% RSLogix 500 project I2P Job 13 B Alexander_Loynd.RSS, saved by version 10.00.00.00 %
PROJECT "ML06A"    % processor: Bul.1763 MicroLogix 1100 Series B %

PROGRAM FILES
  LAD 2   13 rungs

DATA FILES
  O0 OUTPUT  4 elements
  I1 INPUT  6 elements
  S2 STATUS  66 elements
  B3 BINARY  1 elements
  T4 TIMER  1 elements
  C5 COUNTER  1 elements
  R6 CONTROL  1 elements
  N7 INTEGER  1 elements
  F8 FLOAT  1 elements

LADDER 2
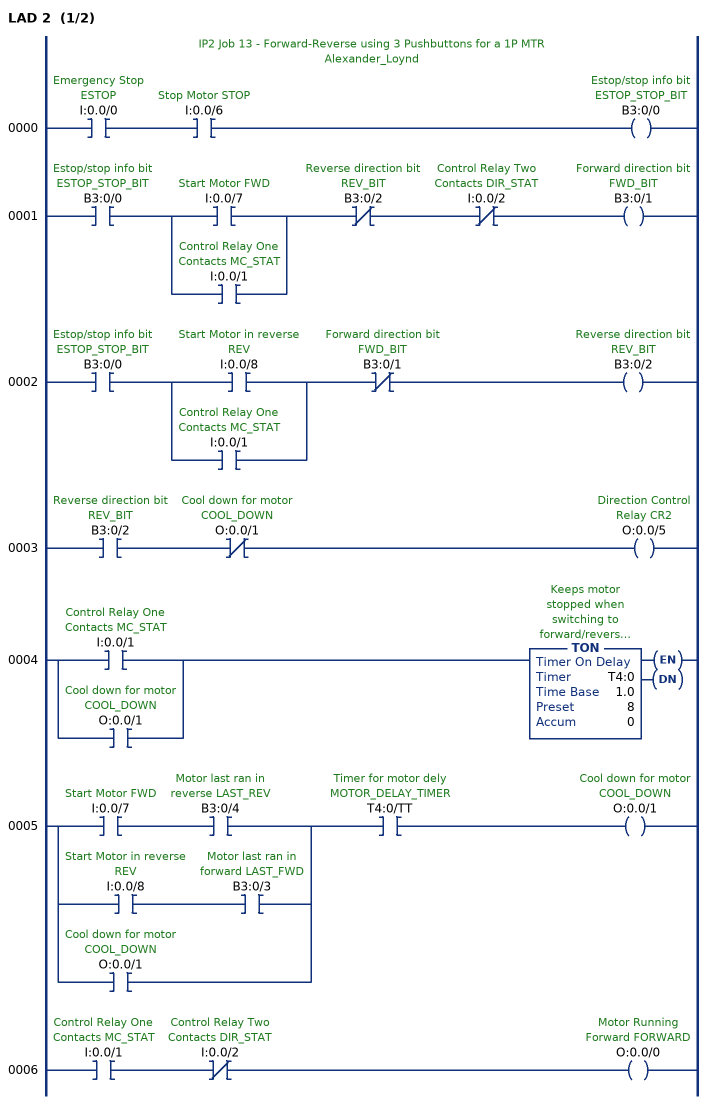
% Rung: 0 %
% IP2 Job 13 - Forward-Reverse using 3 Pushbuttons for a 1P MTR
% Alexander_Loynd %
SOR XIC I:0.0/0 XIC I:0.0/6 OTE B3:0/0 EOR
%   I:0.0/0  ESTOP  "Emergency Stop" %
%   I:0.0/6  STOP  "Stop Motor" %
%   B3:0/0  ESTOP_STOP_BIT  "Estop/stop info bit" %
% Rung: 1 %
SOR XIC B3:0/0 BST XIC I:0.0/7 NXB XIC I:0.0/1 BND XIO B3:0/2 XIO I:0.0/2 OTE B3:0/1 EOR
%   B3:0/0  ESTOP_STOP_BIT  "Estop/stop info bit" %
%   I:0.0/7  FWD  "Start Motor" %
%   I:0.0/1  MC_STAT  "Control Relay One Contacts" %
%   B3:0/2  REV_BIT  "Reverse direction bit" %
%   I:0.0/2  DIR_STAT  "Control Relay Two Contacts" %
%   B3:0/1  FWD_BIT  "Forward direction bit" %
% Rung: 2 %
SOR XIC B3:0/0 BST XIC I:0.0/8 NXB XIC I:0.0/1 BND XIO B3:0/1 OTE B3:0/2 EOR
%   B3:0/0  ESTOP_STOP_BIT  "Estop/stop info bit" %
%   I:0.0/8  REV  "Start Motor in reverse" %
%   I:0.0/1  MC_STAT  "Control Relay One Contacts" %
%   B3:0/1  FWD_BIT  "Forward direction bit" %
%   B3:0/2  REV_BIT  "Reverse direction bit" %
% Rung: 3 %
SOR XIC B3:0/2 XIO O:0.0/1 OTE O:0.0/5 EOR
%   B3:0/2  REV_BIT  "Reverse direction bit" %
%   O:0.0/1  COOL_DOWN  "Cool down for motor" %
%   O:0.0/5  CR2  "Direction Control Relay" %
% Rung: 4 %
SOR BST XIC I:0.0/1 NXB XIC O:0.0/1 BND TON T4:0 1.0 8 0 EOR
%   I:0.0/1  MC_STAT  "Control Relay One Contacts" %
%   O:0.0/1  COOL_DOWN  "Cool down for motor" %
%   T4:0  MTR_DELAY  "Keeps motor stopped when switching to forward/reverse" %
% Rung: 5 %
SOR BST XIC I:0.0/7 XIC B3:0/4 NXB BST XIC I:0.0/8 XIC B3:0/3 NXB XIC O:0.0/1 BND BND XIC T4:0/TT OTE O:0.0/1 EOR
%   I:0.0/7  FWD  "Start Motor" %
%   B3:0/4  LAST_REV  "Motor last ran in reverse" %
%   I:0.0/8  REV  "Start Motor in reverse" %
%   B3:0/3  LAST_FWD  "Motor last ran in forward" %
%   O:0.0/1  COOL_DOWN  "Cool down for motor" %
%   T4:0/TT  MOTOR_DELAY_TIMER  "Timer for motor dely" %
% Rung: 6 %
SOR XIC I:0.0/1 XIO I:0.0/2 OTE O:0.0/0 EOR
%   I:0.0/1  MC_STAT  "Control Relay One Contacts" %
%   I:0.0/2  DIR_STAT  "Control Relay Two Contacts" %
%   O:0.0/0  FORWARD  "Motor Running Forward" %

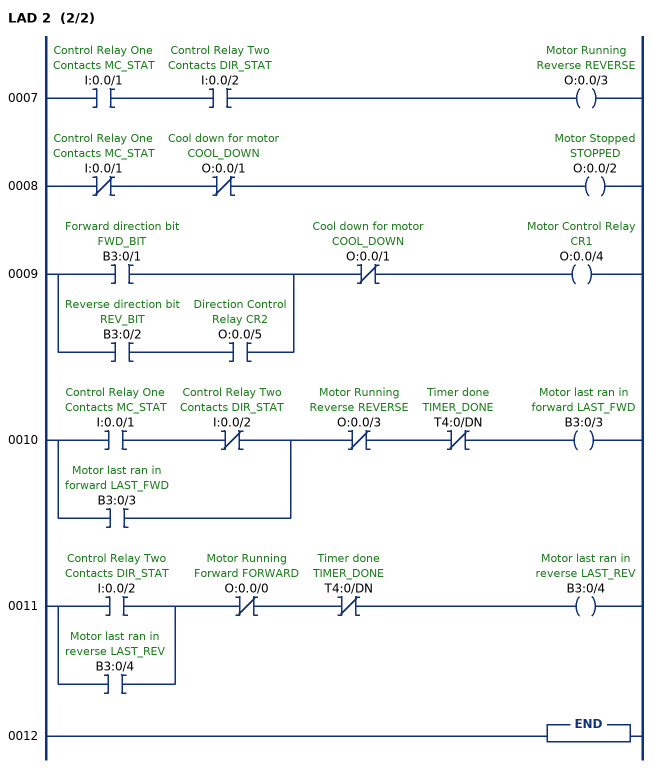
% Rung: 7 %
SOR XIC I:0.0/1 XIC I:0.0/2 OTE O:0.0/3 EOR
%   I:0.0/1  MC_STAT  "Control Relay One Contacts" %
%   I:0.0/2  DIR_STAT  "Control Relay Two Contacts" %
%   O:0.0/3  REVERSE  "Motor Running Reverse" %
% Rung: 8 %
SOR XIO I:0.0/1 XIO O:0.0/1 OTE O:0.0/2 EOR
%   I:0.0/1  MC_STAT  "Control Relay One Contacts" %
%   O:0.0/1  COOL_DOWN  "Cool down for motor" %
%   O:0.0/2  STOPPED  "Motor Stopped" %
% Rung: 9 %
SOR BST XIC B3:0/1 NXB XIC B3:0/2 XIC O:0.0/5 BND XIO O:0.0/1 OTE O:0.0/4 EOR
%   B3:0/1  FWD_BIT  "Forward direction bit" %
%   B3:0/2  REV_BIT  "Reverse direction bit" %
%   O:0.0/5  CR2  "Direction Control Relay" %
%   O:0.0/1  COOL_DOWN  "Cool down for motor" %
%   O:0.0/4  CR1  "Motor Control Relay" %
% Rung: 10 %
SOR BST XIC I:0.0/1 XIO I:0.0/2 NXB XIC B3:0/3 BND XIO O:0.0/3 XIO T4:0/DN OTE B3:0/3 EOR
%   I:0.0/1  MC_STAT  "Control Relay One Contacts" %
%   I:0.0/2  DIR_STAT  "Control Relay Two Contacts" %
%   B3:0/3  LAST_FWD  "Motor last ran in forward" %
%   O:0.0/3  REVERSE  "Motor Running Reverse" %
%   T4:0/DN  TIMER_DONE  "Timer done" %
% Rung: 11 %
SOR BST XIC I:0.0/2 NXB XIC B3:0/4 BND XIO O:0.0/0 XIO T4:0/DN OTE B3:0/4 EOR
%   I:0.0/2  DIR_STAT  "Control Relay Two Contacts" %
%   B3:0/4  LAST_REV  "Motor last ran in reverse" %
%   O:0.0/0  FORWARD  "Motor Running Forward" %
%   T4:0/DN  TIMER_DONE  "Timer done" %
% Rung: 12 %
SOR END EOR

OTHER DOCUMENTED ADDRESSES
  I:0.0/3  DIRECTION_A  "Forward direction 3PSS"
  I:0.0/4  DIRECTION_B  "Reverse direction 3PSS"
  I:0.0/5  2PSS  "Two Position Selector Switch"
  PB1  "Start Motor"

DATA TABLE (non-zero values as saved)
DATA T4
% .PRE .ACC %
% T4:0 % 8 0
